// This function has been automatically generated from the project information.
VAR_GLOBAL CONSTANT
	{attribute 'const_non_replaced'}
	stLibVersion_Base_Elements : ST_LibVersion := (iMajor := 0, iMinor := 0, iBuild := 0, iRevision := 3, sVersion := '0.0.0.3');
END_VAR

(* stored: Version 1.1.0.1, ProductVersion 3.1.0.19
   GVL Global_Version: Id {ed2b94b4-192a-44ca-8117-862238c6523b} *)
